(* IEC 61131-3 sources: Sps24ProgettoDirectLoadingOOP/src/OOP, 5 files *)

(* ---- UserDataType.st ---- *)
NAMESPACE libUdtOop

    TYPE
        gripperInterface : STRUCT
            gripperCmd : gripperCommands;
            gripperOpened : BOOL;
            gripperClosed : BOOL;
        END_STRUCT;
    END_TYPE

    TYPE
        gripperCommands : STRUCT
            openGripper : BOOL;
            closeGripper : BOOL;
        END_STRUCT;
    END_TYPE

    TYPE
        axisInterface : STRUCT
            axisCmd : axisCommands;
            axisOn : BOOL;
            axisReferenced : BOOL;
            axisError : BOOL;
            axisActualPosition : LREAL;
            axisPos1 : BOOL;
            axisPos2 : BOOL;
        END_STRUCT;
    END_TYPE

    TYPE
        axisCommands : STRUCT
            powerAxis : BOOL;
            homingAxis : BOOL;
            goToPos1Axis : BOOL;
            goToPos2Axis : BOOL;
        END_STRUCT;
    END_TYPE

    TYPE
        armInterface : STRUCT
            armCmd : armCommands;
            //armPos1 : BOOL;
            //armPos2 : BOOL;
            endPick : BOOL;
            endPlace : BOOL;
        END_STRUCT;
    END_TYPE

    TYPE
        armCommands : STRUCT
            pickArm : BOOL;
            placeArm : BOOL;
        END_STRUCT;
    END_TYPE

    TYPE
        POSITION : LREAL (
            NONE := 0,
            ARMPOS1 := 5.0,
            ARMPOS2 := 100.0,
            BUFFERPOS1 := 270.0,
            BUFFERPOS2 := 90.0,
            TOL := 0.5
        ) := NONE;
    END_TYPE
    TYPE
        DIRECTION : INT (
            DEFAULT := 3,
            STARTMODE := 1
        ) := DEFAULT;
    END_TYPE

    TYPE
        TIMER : LTIME (
            GRIPPER := LT#1s,
            WIP := LT#2s
        ) := GRIPPER;
    END_TYPE

END_NAMESPACE

(* ---- Arm.st ---- *)
USING libUdtOop;
USING Siemens.Simatic.S71500.MotionControl.Native;

NAMESPACE libMotOop

    CLASS PUBLIC ArmClass EXTENDS AxisClass
        {S7.extern=ReadWrite}
        {OpcUa=ReadWrite}
        VAR PUBLIC
            _instGripper : GripperClass;
            _armInterface : armInterface;
            _statePick : INT;
            _statePlace :INT;
        END_VAR

        METHOD PUBLIC Pick
            VAR
                state : INT;
            END_VAR

            //Logica Presa Braccio
            CASE _statePick OF
                0: // Avvio Missione Prendi
                    _armInterface.endPick := FALSE;
                    _statePick := 2;
                2: // La pinza è aperta?
                    IF _instGripper._gripperInterface.gripperOpened THEN
                        _statePick := 4;
                    ELSE
                        _instGripper.OpenGripper(timerGripper := TIMER#GRIPPER);
                    END_IF;
                4: //Vai a posizione di presa (bassa)
                    IF _axisInterface.axisPos1 THEN
                        _statePick := 6;
                    ELSE
                        THIS.MoveAbs(direction := DIRECTION#DEFAULT, position := POSITION#ARMPOS1);
                    END_IF;
                6: //Chiudi la pinza
                    IF _instGripper._gripperInterface.gripperClosed THEN
                        _statePick := 8;
                    ELSE
                        _instGripper.CloseGripper(timerGripper := TIMER#GRIPPER);
                    END_IF;
                8: //Vai a posizione di attesa (alta)
                    IF _axisInterface.axisPos2 THEN
                        _statePick := 0;
                        _armInterface.endPick := TRUE;
                    ELSE
                        THIS.MoveAbs(direction := DIRECTION#DEFAULT, position := POSITION#ARMPOS2);
                    END_IF;
            END_CASE;
        END_METHOD

        METHOD PUBLIC Place
            VAR_OUTPUT
                state : INT;
            END_VAR
            //Logica Posa Braccio
            CASE _statePlace OF
                0: // Avvio Missione Posa
                    _armInterface.endPlace := FALSE;
                    _statePlace := 2;
                2: //Vai a posizione di posa (bassa)
                    IF _axisInterface.axisPos1 THEN
                        _statePlace := 4;
                    ELSE
                        THIS.MoveAbs(direction := DIRECTION#DEFAULT, position := POSITION#ARMPOS1);
                    END_IF;
                4: //Apri la pinza
                    IF _instGripper._gripperInterface.gripperOpened THEN
                        _statePlace := 6;
                    ELSE
                        _instGripper.OpenGripper(timerGripper := TIMER#GRIPPER);
                    END_IF;
                6: //Vai a posizione di attesa (alta)
                    IF _axisInterface.axisPos2 THEN
                        _statePlace := 0;
                        _armInterface.endPlace := TRUE;
                    ELSE
                        THIS.MoveAbs(direction := DIRECTION#DEFAULT, position := POSITION#ARMPOS2);
                    END_IF;
            END_CASE;
        END_METHOD
    END_CLASS

END_NAMESPACE

(* ---- Axis.st ---- *)
USING libUdtOop;
USING Siemens.Simatic.S71500.MotionControl.Native;

NAMESPACE libMotOop

    CLASS PUBLIC AxisClass
        VAR PROTECTED
            _instMcPower : MC_Power;
            _instMcHome : MC_Home;
            _instMcMoveAbs : MC_MoveAbsolute;
            _instMcStop : MC_Stop;
            _axisDB : DB_ANY;
        END_VAR

        {S7.extern=ReadWrite}
        {OpcUa=ReadWrite}
        VAR PUBLIC
            _axisInterface : axisInterface;
        END_VAR

        METHOD PUBLIC SetAxis : BOOL //Init: controllo se gli oggetti tecnologici sono compatibili
            VAR_INPUT
                axisDB : DB_ANY;
            END_VAR
            VAR_TEMP
                _axisAsPos : REF_TO TO_PositioningAxis;
            END_VAR
            _axisDB := axisDB;
            _axisAsPos := AsPositioningAxisRef(_axisDB);
            SetAxis := _axisAsPos <> NULL;
        END_METHOD

        METHOD PUBLIC Power : BOOL //Abilitazione Asse
            VAR_INPUT
                startMode : INT;
            END_VAR
            _instMcPower.StartMode := startMode;
            _instMcPower.Enable := TRUE;
            Power := _instMcPower.Status;
        END_METHOD

        METHOD PUBLIC Homing //Homing Asse
            _instMcHome.Execute := TRUE;
        END_METHOD

        METHOD PUBLIC Stop //Stop Asse
            _instMcStop.Execute := TRUE;
            _instMcStop.Mode := 0;
        END_METHOD

        METHOD PUBLIC MoveAbs //Movimento Asse in posizione
            VAR_INPUT
                direction : INT;
                position : LREAL;
            END_VAR
            _instMcMoveAbs.Execute := TRUE;
            _instMcMoveAbs.Position := position;
            _instMcMoveAbs.Velocity := 25.0;
            _instMcMoveAbs.Direction := direction;
        END_METHOD

        METHOD PUBLIC CyclicCall //Metodo che inizializza le istruzioni di Motion e lo stato dell'Asse
            THIS.CallMcBlocksPosAxis();
        END_METHOD

        METHOD PROTECTED CallMcBlocksPosAxis //Metodo Protetto, non direttamente accessibile
            VAR_TEMP
                _axisAsPos : REF_TO TO_PositioningAxis;
            END_VAR
            _axisAsPos := AsPositioningAxisRef(_axisDB);
            IF _axisAsPos = NULL THEN
                RETURN;
            ELSE
                _instMcPower(Axis := _axisAsPos^);
                _instMcHome(Axis := _axisAsPos^);
                _instMcMoveAbs(Axis := _axisAsPos^);
                _instMcStop(Axis := _axisAsPos^);

                //Gestione Home
                IF _instMcHome.Done THEN
                    _instMcHome.Execute := FALSE;
                END_IF;

                //Gestione Stop
                IF _instMcStop.Done THEN
                    _instMcStop.Execute := FALSE;
                END_IF;

                //Gestione Move
                IF _instMcMoveAbs.Done OR _instMcMoveAbs.CommandAborted THEN
                    _instMcMoveAbs.Execute := FALSE;
                END_IF;

                _axisInterface.axisOn := _instMcPower.Status;
                _axisInterface.axisReferenced := _axisAsPos^.StatusWord.%X5;
                _axisInterface.axisError := _instMcPower.Error OR _instMcHome.Error OR _instMcMoveAbs.Error;
                _axisInterface.axisActualPosition := _axisAsPos^.ActualPosition;
            END_IF;
        END_METHOD

        METHOD PUBLIC CalculatePosition
            VAR_INPUT
                limit1 : LREAL;
                limit2 : LREAL;
            END_VAR
            VAR_TEMP
                _axisAsPos : REF_TO TO_PositioningAxis;
            END_VAR
            _axisAsPos := AsPositioningAxisRef(_axisDB);
            IF _axisAsPos = NULL THEN
                RETURN;
            ELSE
                IF ((limit1 - POSITION#TOL) < _axisAsPos^.ActualPosition) AND (_axisAsPos^.ActualPosition < (limit1 + POSITION#TOL)) THEN
                    _axisInterface.axisPos1 := TRUE;
                ELSE
                    _axisInterface.axisPos1 := FALSE;
                END_IF;
                IF ((limit2 - POSITION#TOL) < _axisAsPos^.ActualPosition) AND (_axisAsPos^.ActualPosition < (limit2 + POSITION#TOL)) THEN
                    _axisInterface.axisPos2 := TRUE;
                ELSE
                    _axisInterface.axisPos2 := FALSE;
                END_IF;
            END_IF;
        END_METHOD
    END_CLASS

END_NAMESPACE

(* ---- Controller.st ---- *)
USING libUdtOop;
USING System.Timer;
USING Siemens.Simatic.S71500.MotionControl.Native;
USING System.EdgeDetection;

NAMESPACE libMotOop

    FUNCTION_BLOCK controlloreCentrale
        VAR_INPUT
            start : BOOL;
            posAxisRot : DB_ANY;
            posAxisRight : DB_ANY;
            posAxisLeft : DB_ANY;
            stop : BOOL;
        END_VAR
        VAR_OUTPUT
            cicloAutomatico : BOOL;
            numeroCicli : INT;
            state : INT;
        END_VAR
        VAR
            timer1 : OnDelay;
            timer2 : OnDelay;
            fallingStop : FallingEdge;
            risingStop : RisingEdge;
            oldState : INT;
        END_VAR
        VAR_IN_OUT
            asseRot : AxisClass;
            asseDx : ArmClass;
            asseSx : ArmClass;
        END_VAR

        risingStop(signal := stop);
        fallingStop(signal := stop);

        CASE state OF
            0: //one-time setup
                IF start THEN
                    asseRot.SetAxis(posAxisRot);
                    asseDx.SetAxis(posAxisRight);
                    asseSx.SetAxis(posAxisLeft);
                    IF NOT fallingStop.detected THEN
                        state := 1;
                    END_IF;
                END_IF;

                //Gestione Stop
                IF stop THEN
                    asseRot.Stop();
                    asseDx.Stop();
                    asseSx.Stop();
                END_IF;

                IF fallingStop.detected THEN
                    state := oldState;
                END_IF;

            1: //Avvio Sequenza
                IF start THEN
                    state := 100;
                    cicloAutomatico := TRUE;
                    asseDx._armInterface.endPick := FALSE;
                    asseDx._armInterface.endPlace := FALSE;
                    asseSx._armInterface.endPick := FALSE;
                    asseSx._armInterface.endPlace := FALSE;
                END_IF;
            100: // Controllo se gli assi sono accesi
                IF asseRot._axisInterface.axisOn AND asseSx._axisInterface.axisOn AND asseDx._axisInterface.axisOn THEN
                    state := 101;
                ELSE
                    IF NOT asseRot._axisInterface.axisOn THEN
                        asseRot.Power(startMode := DIRECTION#STARTMODE);
                    END_IF;
                    IF NOT asseSx._axisInterface.axisOn THEN
                        asseSx.Power(startMode := DIRECTION#STARTMODE);
                    END_IF;
                    IF NOT asseDx._axisInterface.axisOn THEN
                        asseDx.Power(startMode := DIRECTION#STARTMODE);
                    END_IF;
                END_IF;
            101: //Controllo se gli assi sono referenziati
                IF asseRot._axisInterface.axisReferenced AND asseSx._axisInterface.axisReferenced AND asseDx._axisInterface.axisReferenced THEN
                    state := 2;
                ELSE
                    IF NOT asseRot._axisInterface.axisReferenced THEN
                        asseRot.Homing();
                    END_IF;
                    IF NOT asseSx._axisInterface.axisReferenced THEN
                        asseSx.Homing();
                    END_IF;
                    IF NOT asseDx._axisInterface.axisReferenced THEN
                        asseDx.Homing();
                    END_IF;
                END_IF;
            2: // Ruota AsseRot in Pos 1
                IF asseRot._axisInterface.axisPos1 THEN
                    state := 4;
                ELSE
                    asseRot.MoveAbs(direction := DIRECTION#DEFAULT, position := POSITION#BUFFERPOS1);
                END_IF;
            4: // Prendi con AsseSx
                IF asseSx._armInterface.endPick THEN
                    asseSx._armInterface.endPick := FALSE;
                    state := 6;
                ELSE
                    asseSx.Pick();
                END_IF;
            6: // Attesa
                timer1(signal := TRUE, duration := TIMER#WIP);
                IF timer1.output THEN
                    timer1(signal := FALSE, duration := TIMER#WIP);
                    state := 8;
                END_IF;
            8: // Posa con AsseSx
                IF asseSx._armInterface.endPlace THEN
                    asseSx._armInterface.endPlace := FALSE;
                    state := 10;
                ELSE
                    asseSx.Place();
                END_IF;
            10: // Ruota AsseRot in Pos 2
                IF asseRot._axisInterface.axisPos2 THEN
                    state := 12;
                ELSE
                    asseRot.MoveAbs(direction := DIRECTION#DEFAULT, position := POSITION#BUFFERPOS2);
                END_IF;
            12: // Prendi con AsseDx
                IF asseDx._armInterface.endPick THEN
                    asseDx._armInterface.endPick := FALSE;
                    state := 14;
                ELSE
                    asseDx.Pick();
                END_IF;
            14: //Attesa
                timer2(signal := TRUE, duration := TIMER#WIP);
                IF timer2.output THEN
                    timer2(signal := FALSE, duration := TIMER#WIP);
                    state := 16;
                END_IF;
            16: // Posa con AsseDx
                IF asseDx._armInterface.endPlace THEN
                    asseDx._armInterface.endPlace := FALSE;
                    state := 30;
                ELSE
                    asseDx.Place();
                END_IF;
            30: //Fine Sequenza
                state := 1;
                cicloAutomatico := FALSE;
                numeroCicli := numeroCicli + 1;
        END_CASE;

        asseRot.CyclicCall();
        asseRot.CalculatePosition(POSITION#BUFFERPOS1, POSITION#BUFFERPOS2);
        asseDx.CyclicCall();
        asseDx.CalculatePosition(POSITION#ARMPOS1, POSITION#ARMPOS2);
        asseSx.CyclicCall();
        asseSx.CalculatePosition(POSITION#ARMPOS1, POSITION#ARMPOS2);

        IF risingStop.detected THEN
            oldState := state;
            state := 0;
        END_IF;
    END_FUNCTION_BLOCK

END_NAMESPACE

(* ---- Gripper.st ---- *)
USING libUdtOop;
USING System.Timer;

NAMESPACE libMotOop

    CLASS PUBLIC GripperClass
        VAR PROTECTED
            _instTimerOpen : OnDelay;
            _instTimerClose : OnDelay;
        END_VAR
        VAR PUBLIC
            _gripperInterface : gripperInterface;
        END_VAR

        METHOD PUBLIC OpenGripper
            VAR_INPUT
                timerGripper : LTIME;
            END_VAR
            _gripperInterface.gripperCmd.closeGripper := FALSE;
            _gripperInterface.gripperCmd.openGripper := TRUE;

            _gripperInterface.gripperClosed := FALSE;
            _instTimerOpen(signal := TRUE, duration := timerGripper, output => _gripperInterface.gripperOpened);
        END_METHOD

        METHOD PUBLIC CloseGripper
            VAR_INPUT
                timerGripper : LTIME;
            END_VAR
            _gripperInterface.gripperCmd.openGripper := FALSE;
            _gripperInterface.gripperCmd.closeGripper := TRUE;

            _gripperInterface.gripperOpened := FALSE;
            _instTimerClose(signal := TRUE, duration := timerGripper, output => _gripperInterface.gripperClosed);
        END_METHOD
    END_CLASS

END_NAMESPACE
